SUBAPPLICATION SS3_v_direct_SubApp (* Subapplication Type *)
  (* Standard: 61499-2 *)
  (* Version 1.0, 2024-07-25, DEVIASH *)
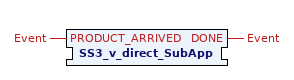
  EVENT_INPUT
    PRODUCT_ARRIVED;
  END_EVENT
  EVENT_OUTPUT
    DONE;
  END_EVENT
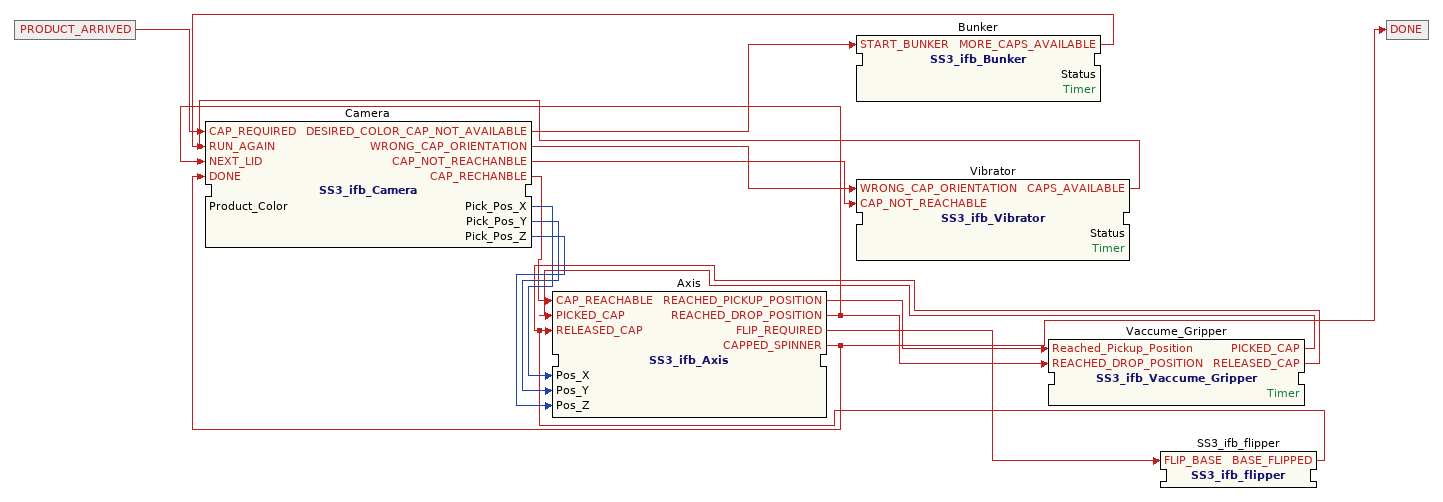
  FBS
    Bunker : SS3_ifb_Bunker;
    Vibrator : SS3_ifb_Vibrator;
    Camera : SS3_ifb_Camera;
    Axis : SS3_ifb_Axis;
    Vaccume_Gripper : SS3_ifb_Vaccume_Gripper;
    SS3_ifb_flipper : SS3_ifb_flipper;
  END_FBS
  EVENT_CONNECTIONS
    Camera.DESIRED_COLOR_CAP_NOT_AVAILABLE TO Bunker.START_BUNKER;
    Bunker.MORE_CAPS_AVAILABLE TO Camera.RUN_AGAIN;
    Camera.WRONG_CAP_ORIENTATION TO Vibrator.WRONG_CAP_ORIENTATION;
    Camera.CAP_NOT_REACHANBLE TO Vibrator.CAP_NOT_REACHABLE;
    Vibrator.CAPS_AVAILABLE TO Camera.RUN_AGAIN;
    Camera.CAP_RECHANBLE TO Axis.CAP_REACHABLE;
    PRODUCT_ARRIVED TO Camera.CAP_REQUIRED;
    Axis.REACHED_PICKUP_POSITION TO Vaccume_Gripper.Reached_Pickup_Position;
    Vaccume_Gripper.PICKED_CAP TO Axis.PICKED_CAP;
    Axis.REACHED_DROP_POSITION TO Vaccume_Gripper.REACHED_DROP_POSITION;
    Vaccume_Gripper.RELEASED_CAP TO Axis.RELEASED_CAP;
    Axis.REACHED_DROP_POSITION TO Camera.NEXT_LID;
    Axis.FLIP_REQUIRED TO SS3_ifb_flipper.FLIP_BASE;
    SS3_ifb_flipper.BASE_FLIPPED TO Axis.RELEASED_CAP;
    Axis.CAPPED_SPINNER TO Camera.DONE;
    Axis.CAPPED_SPINNER TO DONE;
  END_CONNECTIONS
  DATA_CONNECTIONS
    Camera.Pick_Pos_X TO Axis.Pos_X;
    Camera.Pick_Pos_Y TO Axis.Pos_Y;
    Camera.Pick_Pos_Z TO Axis.Pos_Z;
  END_CONNECTIONS
END_SUBAPPLICATION
